// Mitsubishi GX Works2 project: 28   PLC: FX3G

// task Task_01 (event TRUE, interval 0, priority 31): POU_01

PROGRAM POU_01
VAR
  peopleCount : INT;
  wstep : INT;
  ton1 : TON;
  ton2 : TON;
  rt1 : R_TRIG;
  rt2 : R_TRIG;
END_VAR
IF M8002 THEN
	peopleCount := 0;
END_IF;

rt1(_CLK := M2);
rt2(_CLK := M3);

IF rt1.Q THEN
	peopleCount := peopleCount + 1;
END_IF;

IF rt2.Q THEN
	peopleCount := peopleCount - 1;
END_IF;
	
IF (peopleCount > 0) AND M0 THEN
	Y0 := TRUE;
	Y1 := NOT M1;
END_IF;

IF peopleCount <= 0 THEN
	M0 := FALSE;
	M1 := FALSE;
	ton1(IN := TRUE, PT := T#5s);
	IF (ton1.Q) THEN
		Y1 := FALSE;
	END_IF;
	
	ton2(IN := ton1.Q, PT := T#5s);
	IF (ton2.Q) THEN
		Y0 := FALSE;
	END_IF;
ELSE
	ton1(IN := FALSE);
	ton2(IN := FALSE);
END_IF;
END_PROGRAM
